(* CoDeSys 2.3 export: TARAS.EXP *)

(* POU Rooms/Taras, ST *)
FUNCTION_BLOCK Taras
VAR_INPUT
END_VAR
VAR_OUTPUT
END_VAR
VAR
	mainLamp:ButtonTriggeredTimedOnOff:= (timeSetup:= 1200);
END_VAR
mainLamp(input:=S4_1d, output => S12_1);
END_FUNCTION_BLOCK
